PROGRAM PRG_SA_WINDOW
VAR
    xFirstPass		: BOOL;
    fbFSInit		: R_TRIG;

    state			: E_STATES;

    bExtPress : BOOL;

    xExtILK_OK_BLW: INT;

    g_FastFaultOutputNA: FB_HardwareFFOutput;
    g_fbArbiterNA: FB_Arbiter(3);
END_VAR

fbFSInit( CLK := TRUE, Q => xFirstPass);
(* On first PLC pass, put valve into init state*)
IF xFirstPass THEN
    state:= E_STATES.INIT;
    xSAOverrideMode := FALSE;
    SetupMode := FALSE;
END_IF
bExtPress:= qRIXS_SA_GCP_01.PG.xAT_VAC;


//STATE ACTIONS
CASE state OF

 E_STATES.INIT:
        qRIXS_SC_VGC_04.M_Set_OPN_SW(FALSE); //Isolation Valve closed
        qRIXS_SC_VGC_05.M_Set_CLS_SW(FALSE); // Window valve OPEN
        qRIXS_SC_VGC_04.i_xOverrideMode := qRIXS_SC_VGC_05.i_xOverrideMode := FALSE;
        //Transition
        if (qRIXS_SC_VGC_04.M_IsClosed() AND qRIXS_SC_VGC_05.M_IsOpen()) THEN
            state:= E_STATES.NOT_SAFE;
        END_IF

E_STATES.NOT_SAFE: // System is not allowed to actuate, i.e all interlocks are in effect
    qRIXS_SC_VGC_04.M_Set_OPN_SW(qRIXS_SC_VGC_04.iq_stValve.q_xOPN_DO );
     //C_1.i_xExt_OK := VGC_1.i_xEPS_OPN_OK := VGC_1.i_xEPS_CLS_OK:= FALSE;
    qRIXS_SC_VGC_05.i_xExtILK_OK:= FALSE;
    qRIXS_SC_VGC_04.i_xOverrideMode := qRIXS_SC_VGC_05.i_xOverrideMode := FALSE;

    //Transition
    //IF (US_GCC.IG.xAT_VAC AND DS_GCC.IG.xAT_VAC) THEN state:= E_STATES.READY; END_IF
    IF (bExtPress AND qRIXS_SC_GCC_01.IG.xAT_VAC) THEN state:= E_STATES.READY; END_IF



 E_STATES.READY: // OK to MOVE
     // Release the external interlock so the differential pressure inlk is in effect
     qRIXS_SC_VGC_04.i_xExt_OK:= qRIXS_SC_VGC_04.i_xEPS_OK :=TRUE;
    //permission to insert window valve only when US vacuum is good??
    qRIXS_SC_VGC_05.i_xExtILK_OK:= bExtPress;
    // Valves  alternate positions.
    If (qRIXS_SC_VGC_05.M_IsClosed()) THEN  qRIXS_SC_VGC_04.M_Set_OPN_SW(TRUE);
    ELSIF (qRIXS_SC_VGC_05.M_IsOpen()) THEN qRIXS_SC_VGC_04.M_Set_OPN_SW(FALSE);
    END_IF

// bOverride := TRUE;
 E_STATES.OVERRIDE:
    // Override Mode is enabled for all valves
     qRIXS_SC_VGC_04.i_xOverrideMode :=qRIXS_SC_VGC_05.i_xOverrideMode := TRUE;
    // Exit of Override mode always goes back to init
     IF NOT(xSAOverrideMode) THEN state:= E_STATES.INIT; END_IF


 E_STATES.SETUP:
    // Window valve remains retracted
     qRIXS_SC_VGC_05.i_xExtILK_OK := FALSE;
    // Isolation valves operates like standard gate valves
    qRIXS_SC_VGC_04.i_xExt_OK := TRUE;
    // exit to init just to be safe?
    IF NOT(SetupMode) THEN state:= E_STATES.INIT; END_IF
END_CASE


// STATE TRANSITIONS
// the system can go to setup state from any other state except override
IF (SetupMode) AND (state<>E_STATES.OVERRIDE) THEN state:= E_STATES.SETUP;
// the system can go to override state from any other state except setup
ELSIF (xSAOverrideMode) AND (state<>E_STATES.SETUP) THEN state:= E_STATES.OVERRIDE;
//Loss of at vac signal makes the system go to init/not safe to move state
ELSIF (NOT bExtPress) OR (NOT qRIXS_SC_GCC_01.IG.xAT_VAC) THEN state:= E_STATES.INIT;
//ELSIF (NOT US_GCC.IG.xAT_VAC) OR (NOT DS_GCC.IG.xAT_VAC) THEN state:= E_STATES.INIT;
END_IF




qRIXS_SC_VGC_04(
    i_stUSG:= qRIXS_SC_GCC_01.IG ,
    i_stDSG:= qRIXS_SA_GCP_02.PG ,
    i_xDis_DPIlk:= FALSE ,
    i_xPMPS_OK:= TRUE ,
    i_xEPS_OK:= ,
    i_xExt_OK:= ,
    i_xOverrideMode:= ,
    i_xReset:= ,
    i_xIsAperture:= TRUE,
    i_sDevName:= ,
    i_nTransitionRootID:= ,
    iq_stValve=> ,
    xMPS_OK=> ,
    io_fbFFHWO:=g_FastFaultOutputNA,
    fbArbiter:= g_fbArbiterNA
);


qRIXS_SC_VGC_05(
    i_xExtILK_OK:= ,
    i_xOverrideMode:= ,
    iq_stValve=>  );

END_PROGRAM

(* stored: Version 1.1.0.1, ProductVersion 3.1.4022.18
   POU PRG_SA_WINDOW: Id {7abc0b72-bfc7-40b5-9fc5-6d9e0631f363}, SpecialFunc None *)
